{attribute 'OPC.UA.DA.StructuredType' := '1'}
FUNCTION_BLOCK FB_BagFilter EXTENDS FB_BaseDevice IMPLEMENTS I_Device

VAR
	{attribute 'OPC.UA.DA' := '1'}
  	{attribute 'OPC.UA.DA.StructuredType' := '1'}
	fbDiffPress_Upstream: I_Sensor(SensorID := '', SensorDescr := '', SensorType := E_SensorType.Analogue);
	{attribute 'OPC.UA.DA' := '1'}
  	{attribute 'OPC.UA.DA.StructuredType' := '1'}
	fbDiffPress_Downstream: I_Sensor(SensorID := '', SensorDescr := '', SensorType := E_SensorType.Analogue);
	{attribute 'OPC.UA.DA' := '1'}
	nDiffPressure: REAL;
	
END_VAR

VAR_IN_OUT
	{attribute 'OPC.UA.DA' := '1'}
	nMaxPressure: UINT;
END_VAR

// Bag Filters do not actually do anything, however it will be useful to maintain an OEE object for these
// We can then monitor when filters need to be replaced

nDiffPressure := ABS(fbDiffPress_Upstream.getValue() - fbDiffPress_Downstream.getValue());

{warning 'add method implementation '}
METHOD disable : BOOL
END_METHOD

{warning 'add method implementation '}
METHOD enable : BOOL
END_METHOD

METHOD FB_init : BOOL
VAR_INPUT
	bInitRetains : BOOL; // if TRUE, the retain variables are initialized (warm start / cold start)
	bInCopyCode : BOOL;  // if TRUE, the instance afterwards gets moved into the copy code (online change)
	
	FilterID: STRING(80);
	FilterDescr: STRING(255);

END_VAR
sID := FilterID;
sDescr := FilterDescr;
END_METHOD

METHOD getDiffPressure : REAL
VAR_INPUT
END_VAR
//getDiffPressure := fbSensorPIT_Upstream.getValue() - fbSensorPIT_Downstream.getValue();
END_METHOD

METHOD setPressureLimits : BOOL
VAR_INPUT
	PressTx_Upstream: I_Sensor(SensorID := '', SensorDescr := '', SensorType := E_SensorType.Analogue);
	PressTx_Downstream: I_Sensor(SensorID := '', SensorDescr := '', SensorType := E_SensorType.Analogue);
END_VAR

fbDiffPress_Downstream := PressTx_Downstream;
fbDiffPress_Upstream := PressTx_Upstream;
END_METHOD

END_FUNCTION_BLOCK

(* stored: Version 1.1.0.1, ProductVersion 3.1.4024.12
   POU FB_BagFilter: Id {6d60cb67-a8de-4da2-8f63-8e864ca4c6b0}, SpecialFunc None
   Method disable: Id {dd814a7e-ec48-47bf-baf5-14fd1672986b}
   Method enable: Id {1f5586b2-fe22-4267-814e-9ca576b99d19}
   Method FB_init: Id {0ac5faf3-2585-41fe-a3f1-080f9ada033c}
   Method getDiffPressure: Id {f15d7331-6ccc-40fe-ae5d-bb9fe9c4606b}
   Method setPressureLimits: Id {f9e53c89-5043-4bae-bdbf-96455fedcebb} *)
